// TIA Portal V20 export
FUNCTION_BLOCK "Sequence_3_NgPnP"   // FB245, LAD
AUTHOR : ERsystem_FA2_DH. Kim
// stored: IsIECCheckEnabled true, MemoryReserve 100, Namespace Unit1.Em4, SetENOAutomatically false
   VAR
      instSequenceLADStatus { ExternalWritable := 'False'} : "LAF_StatusLadSequence";
      instSequenceLADControl { ExternalWritable := 'False'} : "LAF_ControlLadSequence";
      statTonTime { ExternalWritable := 'False'} : Array[0..9999] of TON_TIME;
   END_VAR
   VAR_TEMP
      tempCustomerAction : Bool;   // Placeholder for possible actions
      tempDo_nothing_and_wait_for_init : Bool;   // Placeholder for doing nothing
      tempSafeStateCondition : Bool;   // Temp Condition for the equipment module to be in a safe state
   END_VAR
   VAR CONSTANT
      delayTime : Time := T#300ms;
      STEP_IDLE : DInt := 1;
      STEP_IMMEDIATE_STOP : DInt := 9001;   // Step executed when an immediate stop command is triggered for the sequence (i.e. when unit is in state aborting)
      JOB_1_STEP_01 : DInt := 101;
      JOB_1_STEP_10 : DInt := 110;
      JOB_1_STEP_20 : DInt := 120;
      JOB_1_STEP_30 : DInt := 130;
      JOB_1_STEP_80 : DInt := 180;
      JOB_1_STEP_81 : DInt := 181;
      JOB_1_STEP_90 : DInt := 190;
      JOB_2_STEP_01 : DInt := 201;
      JOB_2_STEP_10 : DInt := 210;
      JOB_2_STEP_20 : DInt := 220;
      JOB_2_STEP_30 : DInt := 230;
      JOB_2_STEP_31 : DInt := 231;
      JOB_2_STEP_40 : DInt := 240;
      JOB_2_STEP_80 : DInt := 280;
      JOB_2_STEP_90 : DInt := 290;
      JOB_3_STEP_01 : DInt := 301;
      JOB_3_STEP_20 : DInt := 320;
      JOB_3_STEP_30 : DInt := 330;
      JOB_3_STEP_40 : DInt := 340;
      JOB_3_STEP_90 : DInt := 390;
      FALSE : Bool := FALSE;
      TRUE : Bool := TRUE;
   END_VAR
   VAR_TEMP   // added for the SCL form of the ladder/FBD networks
      _w1 : Bool;
   END_VAR
BEGIN

REGION Network 1: BLOCK INFO HEADER
   // (company) / (C) Copyright (year)
   // ---------------------------------------------------------------------------------
   // Title:                             (Title of this block)
   // Comment/Function: (that is implemented in the block)
   // Library/Family:           (that the source is dedicated to)
   // Author:                        (department / person in charge / contact)
   // Target System:          (test system with FW version)
   // Engineering:              TIA Portal (SW version)
   // Restrictions:               (OB types, etc.)
   // Requirements:           (hardware, technological package, etc.)
   // ---------------------------------------------------------------------------------
   // Change log table:
   // Version          | Date             | Signature      | Expert in charge  | Changes applied ------------------------|----------------------|-------------------------|--------------------------------|-----------------------
   // 001.000.000 | yyyy-mm-dd | 0x00000000 | (name of expert) | First released version
END_REGION

REGION Network 2: DESCRIPTION
   // This is a template block provided by the Automation Framework. It can be used to create an own project.
   // The Block Info Header is prepared to put in your own data.
   // Description of the block could be added here and the docu created by Code2Docu.
END_REGION

REGION Network 3: ********************* CONTROL *************************
END_REGION

REGION Network 4: Sequence Control
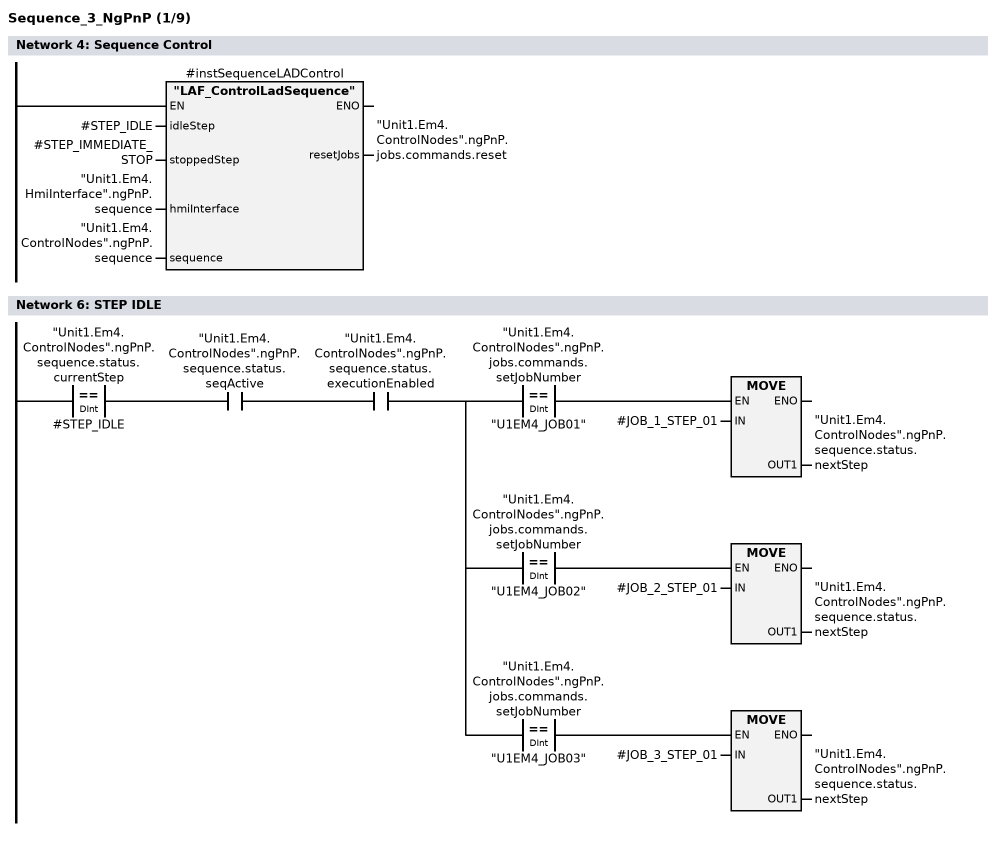
   RUNG wire#powerrail
      #instSequenceLADControl(idleStep := #STEP_IDLE, stoppedStep := #STEP_IMMEDIATE_STOP, hmiInterface := "Unit1.Em4.HmiInterface".ngPnP.sequence, sequence := "Unit1.Em4.ControlNodes".ngPnP.sequence, resetJobs => "Unit1.Em4.ControlNodes".ngPnP.jobs.commands.reset)
   END_RUNG
   // the same network as SCL:
   #instSequenceLADControl(idleStep := #STEP_IDLE,   // "LAF_ControlLadSequence"
                           stoppedStep := #STEP_IMMEDIATE_STOP,
                           hmiInterface := "Unit1.Em4.HmiInterface".ngPnP.sequence,
                           sequence := "Unit1.Em4.ControlNodes".ngPnP.sequence,
                           resetJobs => "Unit1.Em4.ControlNodes".ngPnP.jobs.commands.reset);
END_REGION

REGION Network 5: *************** JOB SELECT **************************
END_REGION

REGION Network 6: STEP IDLE
   RUNG wire#powerrail
      { S7_Templates := "SrcType := DInt" } EQ_Contact(in1 := "Unit1.Em4.ControlNodes".ngPnP.sequence.status.currentStep, in2 := #STEP_IDLE)
      Contact( "Unit1.Em4.ControlNodes".ngPnP.sequence.status.seqActive )
      Contact( "Unit1.Em4.ControlNodes".ngPnP.sequence.status.executionEnabled )
      wire#w1
      { S7_Templates := "SrcType := DInt" } EQ_Contact(in1 := "Unit1.Em4.ControlNodes".ngPnP.jobs.commands.setJobNumber, in2 := "U1EM4_JOB01")
      Move(in := #JOB_1_STEP_01, out1 => "Unit1.Em4.ControlNodes".ngPnP.sequence.status.nextStep)
   END_RUNG
   RUNG wire#w1
      { S7_Templates := "SrcType := DInt" } EQ_Contact(in1 := "Unit1.Em4.ControlNodes".ngPnP.jobs.commands.setJobNumber, in2 := "U1EM4_JOB02")
      Move(in := #JOB_2_STEP_01, out1 => "Unit1.Em4.ControlNodes".ngPnP.sequence.status.nextStep)
   END_RUNG
   RUNG wire#w1
      { S7_Templates := "SrcType := DInt" } EQ_Contact(in1 := "Unit1.Em4.ControlNodes".ngPnP.jobs.commands.setJobNumber, in2 := "U1EM4_JOB03")
      Move(in := #JOB_3_STEP_01, out1 => "Unit1.Em4.ControlNodes".ngPnP.sequence.status.nextStep)
   END_RUNG
   // the same network as SCL:
   #_w1 := ("Unit1.Em4.ControlNodes".ngPnP.sequence.status.currentStep = #STEP_IDLE) AND "Unit1.Em4.ControlNodes".ngPnP.sequence.status.seqActive AND "Unit1.Em4.ControlNodes".ngPnP.sequence.status.executionEnabled;
   IF #_w1 AND ("Unit1.Em4.ControlNodes".ngPnP.jobs.commands.setJobNumber = "U1EM4_JOB01") THEN
       "Unit1.Em4.ControlNodes".ngPnP.sequence.status.nextStep := #JOB_1_STEP_01;
   END_IF;
   IF #_w1 AND ("Unit1.Em4.ControlNodes".ngPnP.jobs.commands.setJobNumber = "U1EM4_JOB02") THEN
       "Unit1.Em4.ControlNodes".ngPnP.sequence.status.nextStep := #JOB_2_STEP_01;
   END_IF;
   IF #_w1 AND ("Unit1.Em4.ControlNodes".ngPnP.jobs.commands.setJobNumber = "U1EM4_JOB03") THEN
       "Unit1.Em4.ControlNodes".ngPnP.sequence.status.nextStep := #JOB_3_STEP_01;
   END_IF;
END_REGION

REGION Network 7: *************** JOB[1] EM HOMING ************************
END_REGION

REGION Network 8: Step[101] : JOB[1] Condition
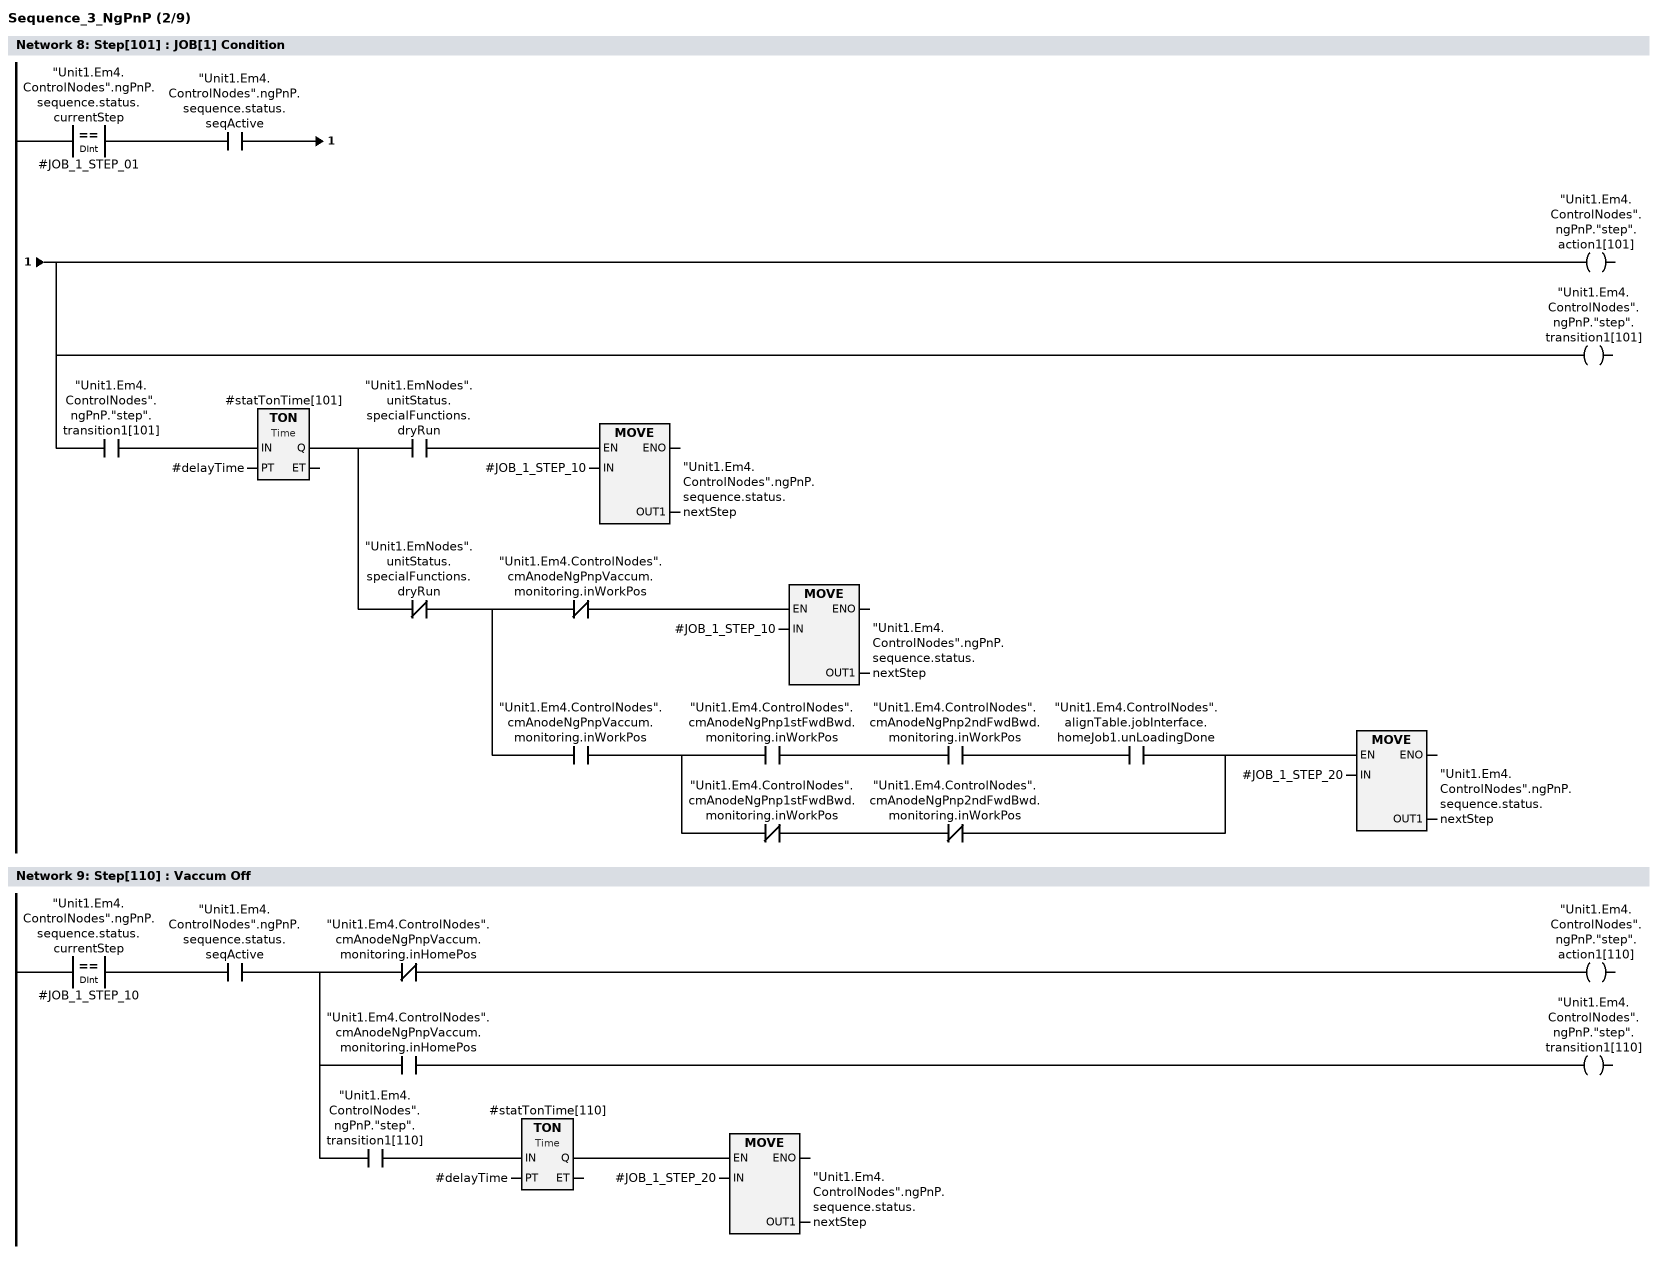
   RUNG wire#powerrail
      { S7_Templates := "SrcType := DInt" } EQ_Contact(in1 := "Unit1.Em4.ControlNodes".ngPnP.sequence.status.currentStep, in2 := #JOB_1_STEP_01)
      Contact( "Unit1.Em4.ControlNodes".ngPnP.sequence.status.seqActive )
      wire#w1
      Coil( "Unit1.Em4.ControlNodes".ngPnP."step".action1[101] )
   END_RUNG
   RUNG wire#w1
      Coil( "Unit1.Em4.ControlNodes".ngPnP."step".transition1[101] )
   END_RUNG
   RUNG wire#w1
      Contact( "Unit1.Em4.ControlNodes".ngPnP."step".transition1[101] )
      { S7_Templates := "time_type := Time" } #statTonTime[101].TON(pt := #delayTime, et =>)
      wire#w2
      Contact( "Unit1.EmNodes".unitStatus.specialFunctions.dryRun )
      Move(in := #JOB_1_STEP_10, out1 => "Unit1.Em4.ControlNodes".ngPnP.sequence.status.nextStep)
   END_RUNG
   RUNG wire#w2
      I_Contact( "Unit1.EmNodes".unitStatus.specialFunctions.dryRun )
      wire#w3
      I_Contact( "Unit1.Em4.ControlNodes".cmAnodeNgPnpVaccum.monitoring.inWorkPos )
      Move(in := #JOB_1_STEP_10, out1 => "Unit1.Em4.ControlNodes".ngPnP.sequence.status.nextStep)
   END_RUNG
   RUNG wire#w3
      Contact( "Unit1.Em4.ControlNodes".cmAnodeNgPnpVaccum.monitoring.inWorkPos )
      wire#w4
      Contact( "Unit1.Em4.ControlNodes".cmAnodeNgPnp1stFwdBwd.monitoring.inWorkPos )
      Contact( "Unit1.Em4.ControlNodes".cmAnodeNgPnp2ndFwdBwd.monitoring.inWorkPos )
      Contact( "Unit1.Em4.ControlNodes".alignTable.jobInterface.homeJob1.unLoadingDone )
      wire#w5
      Move(in := #JOB_1_STEP_20, out1 => "Unit1.Em4.ControlNodes".ngPnP.sequence.status.nextStep)
   END_RUNG
   RUNG wire#w4
      I_Contact( "Unit1.Em4.ControlNodes".cmAnodeNgPnp1stFwdBwd.monitoring.inWorkPos )
      I_Contact( "Unit1.Em4.ControlNodes".cmAnodeNgPnp2ndFwdBwd.monitoring.inWorkPos )
   END_RUNG wire#w5
   // the same network as SCL:
   "Unit1.Em4.ControlNodes".ngPnP."step".action1[101] := ("Unit1.Em4.ControlNodes".ngPnP.sequence.status.currentStep = #JOB_1_STEP_01) AND "Unit1.Em4.ControlNodes".ngPnP.sequence.status.seqActive;
   "Unit1.Em4.ControlNodes".ngPnP."step".transition1[101] := ("Unit1.Em4.ControlNodes".ngPnP.sequence.status.currentStep = #JOB_1_STEP_01) AND "Unit1.Em4.ControlNodes".ngPnP.sequence.status.seqActive;
   #statTonTime[101].TON(IN := ("Unit1.Em4.ControlNodes".ngPnP.sequence.status.currentStep = #JOB_1_STEP_01) AND "Unit1.Em4.ControlNodes".ngPnP.sequence.status.seqActive AND "Unit1.Em4.ControlNodes".ngPnP."step".transition1[101],
                         PT := #delayTime);
   IF #statTonTime[101].Q AND "Unit1.EmNodes".unitStatus.specialFunctions.dryRun THEN
       "Unit1.Em4.ControlNodes".ngPnP.sequence.status.nextStep := #JOB_1_STEP_10;
   END_IF;
   #_w1 := #statTonTime[101].Q AND NOT "Unit1.EmNodes".unitStatus.specialFunctions.dryRun;
   IF #_w1 AND NOT "Unit1.Em4.ControlNodes".cmAnodeNgPnpVaccum.monitoring.inWorkPos THEN
       "Unit1.Em4.ControlNodes".ngPnP.sequence.status.nextStep := #JOB_1_STEP_10;
   END_IF;
   IF #_w1 AND "Unit1.Em4.ControlNodes".cmAnodeNgPnpVaccum.monitoring.inWorkPos AND (("Unit1.Em4.ControlNodes".cmAnodeNgPnp1stFwdBwd.monitoring.inWorkPos AND "Unit1.Em4.ControlNodes".cmAnodeNgPnp2ndFwdBwd.monitoring.inWorkPos AND "Unit1.Em4.ControlNodes".alignTable.jobInterface.homeJob1.unLoadingDone) OR (NOT "Unit1.Em4.ControlNodes".cmAnodeNgPnp1stFwdBwd.monitoring.inWorkPos AND NOT "Unit1.Em4.ControlNodes".cmAnodeNgPnp2ndFwdBwd.monitoring.inWorkPos)) THEN
       "Unit1.Em4.ControlNodes".ngPnP.sequence.status.nextStep := #JOB_1_STEP_20;
   END_IF;
END_REGION

REGION Network 9: Step[110] : Vaccum Off
   RUNG wire#powerrail
      { S7_Templates := "SrcType := DInt" } EQ_Contact(in1 := "Unit1.Em4.ControlNodes".ngPnP.sequence.status.currentStep, in2 := #JOB_1_STEP_10)
      Contact( "Unit1.Em4.ControlNodes".ngPnP.sequence.status.seqActive )
      wire#w1
      I_Contact( "Unit1.Em4.ControlNodes".cmAnodeNgPnpVaccum.monitoring.inHomePos )
      Coil( "Unit1.Em4.ControlNodes".ngPnP."step".action1[110] )
   END_RUNG
   RUNG wire#w1
      Contact( "Unit1.Em4.ControlNodes".cmAnodeNgPnpVaccum.monitoring.inHomePos )
      Coil( "Unit1.Em4.ControlNodes".ngPnP."step".transition1[110] )
   END_RUNG
   RUNG wire#w1
      Contact( "Unit1.Em4.ControlNodes".ngPnP."step".transition1[110] )
      { S7_Templates := "time_type := Time" } #statTonTime[110].TON(pt := #delayTime, et =>)
      Move(in := #JOB_1_STEP_20, out1 => "Unit1.Em4.ControlNodes".ngPnP.sequence.status.nextStep)
   END_RUNG
   // the same network as SCL:
   #_w1 := ("Unit1.Em4.ControlNodes".ngPnP.sequence.status.currentStep = #JOB_1_STEP_10) AND "Unit1.Em4.ControlNodes".ngPnP.sequence.status.seqActive;
   "Unit1.Em4.ControlNodes".ngPnP."step".action1[110] := #_w1 AND NOT "Unit1.Em4.ControlNodes".cmAnodeNgPnpVaccum.monitoring.inHomePos;
   "Unit1.Em4.ControlNodes".ngPnP."step".transition1[110] := #_w1 AND "Unit1.Em4.ControlNodes".cmAnodeNgPnpVaccum.monitoring.inHomePos;
   #statTonTime[110].TON(IN := #_w1 AND "Unit1.Em4.ControlNodes".ngPnP."step".transition1[110],
                         PT := #delayTime);
   IF #statTonTime[110].Q THEN
       "Unit1.Em4.ControlNodes".ngPnP.sequence.status.nextStep := #JOB_1_STEP_20;
   END_IF;
END_REGION

REGION Network 10: Step[120] : NG P&P Up
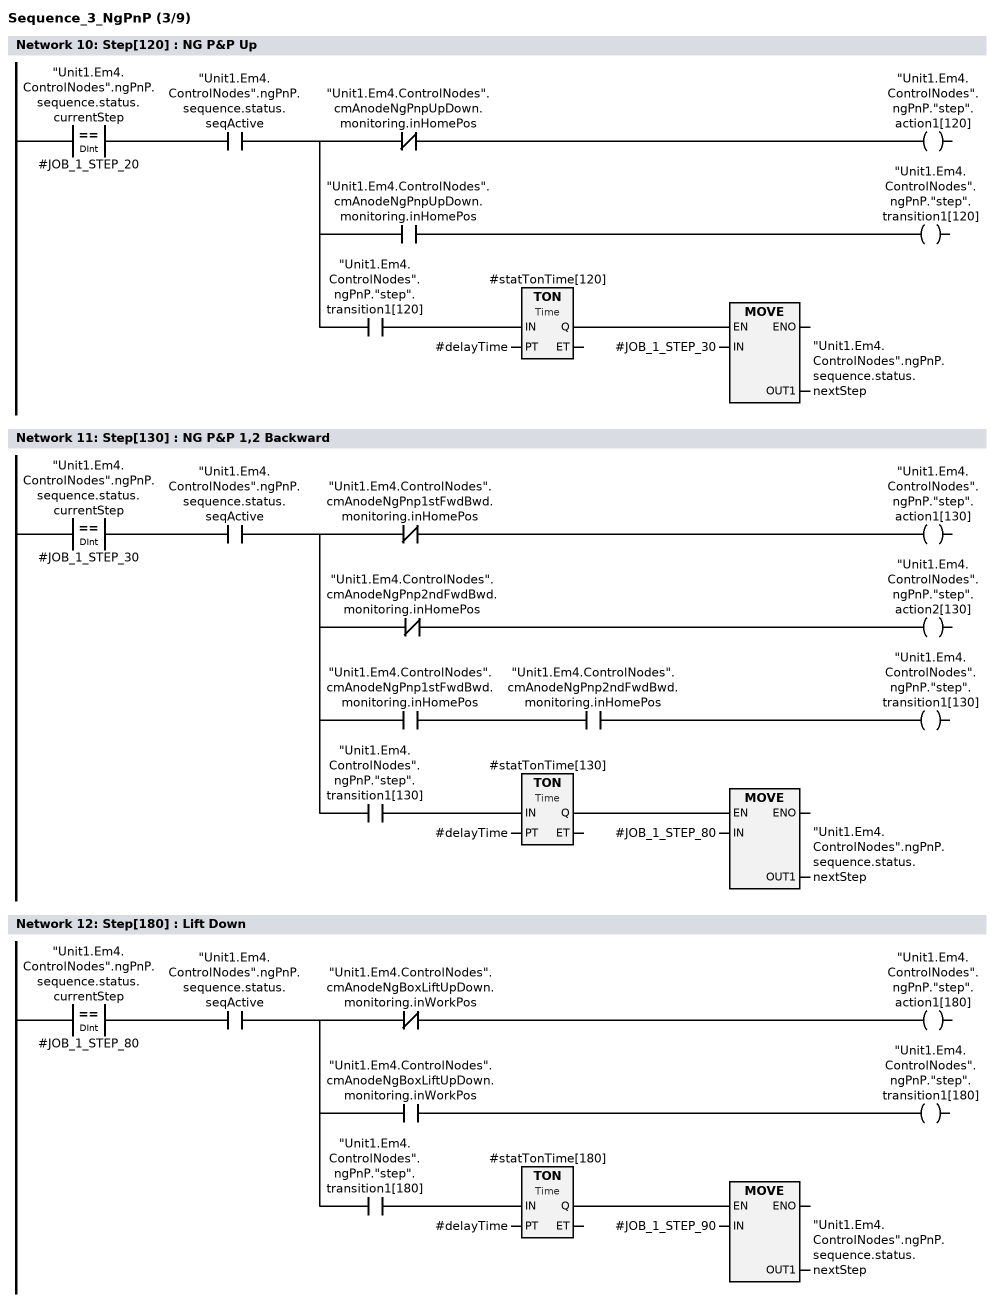
   RUNG wire#powerrail
      { S7_Templates := "SrcType := DInt" } EQ_Contact(in1 := "Unit1.Em4.ControlNodes".ngPnP.sequence.status.currentStep, in2 := #JOB_1_STEP_20)
      Contact( "Unit1.Em4.ControlNodes".ngPnP.sequence.status.seqActive )
      wire#w1
      I_Contact( "Unit1.Em4.ControlNodes".cmAnodeNgPnpUpDown.monitoring.inHomePos )
      Coil( "Unit1.Em4.ControlNodes".ngPnP."step".action1[120] )
   END_RUNG
   RUNG wire#w1
      Contact( "Unit1.Em4.ControlNodes".cmAnodeNgPnpUpDown.monitoring.inHomePos )
      Coil( "Unit1.Em4.ControlNodes".ngPnP."step".transition1[120] )
   END_RUNG
   RUNG wire#w1
      Contact( "Unit1.Em4.ControlNodes".ngPnP."step".transition1[120] )
      { S7_Templates := "time_type := Time" } #statTonTime[120].TON(pt := #delayTime, et =>)
      Move(in := #JOB_1_STEP_30, out1 => "Unit1.Em4.ControlNodes".ngPnP.sequence.status.nextStep)
   END_RUNG
   // the same network as SCL:
   #_w1 := ("Unit1.Em4.ControlNodes".ngPnP.sequence.status.currentStep = #JOB_1_STEP_20) AND "Unit1.Em4.ControlNodes".ngPnP.sequence.status.seqActive;
   "Unit1.Em4.ControlNodes".ngPnP."step".action1[120] := #_w1 AND NOT "Unit1.Em4.ControlNodes".cmAnodeNgPnpUpDown.monitoring.inHomePos;
   "Unit1.Em4.ControlNodes".ngPnP."step".transition1[120] := #_w1 AND "Unit1.Em4.ControlNodes".cmAnodeNgPnpUpDown.monitoring.inHomePos;
   #statTonTime[120].TON(IN := #_w1 AND "Unit1.Em4.ControlNodes".ngPnP."step".transition1[120],
                         PT := #delayTime);
   IF #statTonTime[120].Q THEN
       "Unit1.Em4.ControlNodes".ngPnP.sequence.status.nextStep := #JOB_1_STEP_30;
   END_IF;
END_REGION

REGION Network 11: Step[130] : NG P&P 1,2 Backward
   RUNG wire#powerrail
      { S7_Templates := "SrcType := DInt" } EQ_Contact(in1 := "Unit1.Em4.ControlNodes".ngPnP.sequence.status.currentStep, in2 := #JOB_1_STEP_30)
      Contact( "Unit1.Em4.ControlNodes".ngPnP.sequence.status.seqActive )
      wire#w1
      I_Contact( "Unit1.Em4.ControlNodes".cmAnodeNgPnp1stFwdBwd.monitoring.inHomePos )
      Coil( "Unit1.Em4.ControlNodes".ngPnP."step".action1[130] )
   END_RUNG
   RUNG wire#w1
      I_Contact( "Unit1.Em4.ControlNodes".cmAnodeNgPnp2ndFwdBwd.monitoring.inHomePos )
      Coil( "Unit1.Em4.ControlNodes".ngPnP."step".action2[130] )
   END_RUNG
   RUNG wire#w1
      Contact( "Unit1.Em4.ControlNodes".cmAnodeNgPnp1stFwdBwd.monitoring.inHomePos )
      Contact( "Unit1.Em4.ControlNodes".cmAnodeNgPnp2ndFwdBwd.monitoring.inHomePos )
      Coil( "Unit1.Em4.ControlNodes".ngPnP."step".transition1[130] )
   END_RUNG
   RUNG wire#w1
      Contact( "Unit1.Em4.ControlNodes".ngPnP."step".transition1[130] )
      { S7_Templates := "time_type := Time" } #statTonTime[130].TON(pt := #delayTime, et =>)
      Move(in := #JOB_1_STEP_80, out1 => "Unit1.Em4.ControlNodes".ngPnP.sequence.status.nextStep)
   END_RUNG
   // the same network as SCL:
   #_w1 := ("Unit1.Em4.ControlNodes".ngPnP.sequence.status.currentStep = #JOB_1_STEP_30) AND "Unit1.Em4.ControlNodes".ngPnP.sequence.status.seqActive;
   "Unit1.Em4.ControlNodes".ngPnP."step".action1[130] := #_w1 AND NOT "Unit1.Em4.ControlNodes".cmAnodeNgPnp1stFwdBwd.monitoring.inHomePos;
   "Unit1.Em4.ControlNodes".ngPnP."step".action2[130] := #_w1 AND NOT "Unit1.Em4.ControlNodes".cmAnodeNgPnp2ndFwdBwd.monitoring.inHomePos;
   "Unit1.Em4.ControlNodes".ngPnP."step".transition1[130] := #_w1 AND "Unit1.Em4.ControlNodes".cmAnodeNgPnp1stFwdBwd.monitoring.inHomePos AND "Unit1.Em4.ControlNodes".cmAnodeNgPnp2ndFwdBwd.monitoring.inHomePos;
   #statTonTime[130].TON(IN := #_w1 AND "Unit1.Em4.ControlNodes".ngPnP."step".transition1[130],
                         PT := #delayTime);
   IF #statTonTime[130].Q THEN
       "Unit1.Em4.ControlNodes".ngPnP.sequence.status.nextStep := #JOB_1_STEP_80;
   END_IF;
END_REGION

REGION Network 12: Step[180] : Lift Down
   RUNG wire#powerrail
      { S7_Templates := "SrcType := DInt" } EQ_Contact(in1 := "Unit1.Em4.ControlNodes".ngPnP.sequence.status.currentStep, in2 := #JOB_1_STEP_80)
      Contact( "Unit1.Em4.ControlNodes".ngPnP.sequence.status.seqActive )
      wire#w1
      I_Contact( "Unit1.Em4.ControlNodes".cmAnodeNgBoxLiftUpDown.monitoring.inWorkPos )
      Coil( "Unit1.Em4.ControlNodes".ngPnP."step".action1[180] )
   END_RUNG
   RUNG wire#w1
      Contact( "Unit1.Em4.ControlNodes".cmAnodeNgBoxLiftUpDown.monitoring.inWorkPos )
      Coil( "Unit1.Em4.ControlNodes".ngPnP."step".transition1[180] )
   END_RUNG
   RUNG wire#w1
      Contact( "Unit1.Em4.ControlNodes".ngPnP."step".transition1[180] )
      { S7_Templates := "time_type := Time" } #statTonTime[180].TON(pt := #delayTime, et =>)
      Move(in := #JOB_1_STEP_90, out1 => "Unit1.Em4.ControlNodes".ngPnP.sequence.status.nextStep)
   END_RUNG
   // the same network as SCL:
   #_w1 := ("Unit1.Em4.ControlNodes".ngPnP.sequence.status.currentStep = #JOB_1_STEP_80) AND "Unit1.Em4.ControlNodes".ngPnP.sequence.status.seqActive;
   "Unit1.Em4.ControlNodes".ngPnP."step".action1[180] := #_w1 AND NOT "Unit1.Em4.ControlNodes".cmAnodeNgBoxLiftUpDown.monitoring.inWorkPos;
   "Unit1.Em4.ControlNodes".ngPnP."step".transition1[180] := #_w1 AND "Unit1.Em4.ControlNodes".cmAnodeNgBoxLiftUpDown.monitoring.inWorkPos;
   #statTonTime[180].TON(IN := #_w1 AND "Unit1.Em4.ControlNodes".ngPnP."step".transition1[180],
                         PT := #delayTime);
   IF #statTonTime[180].Q THEN
       "Unit1.Em4.ControlNodes".ngPnP.sequence.status.nextStep := #JOB_1_STEP_90;
   END_IF;
END_REGION

REGION Network 13: Step[190] : JOB[1] Step End
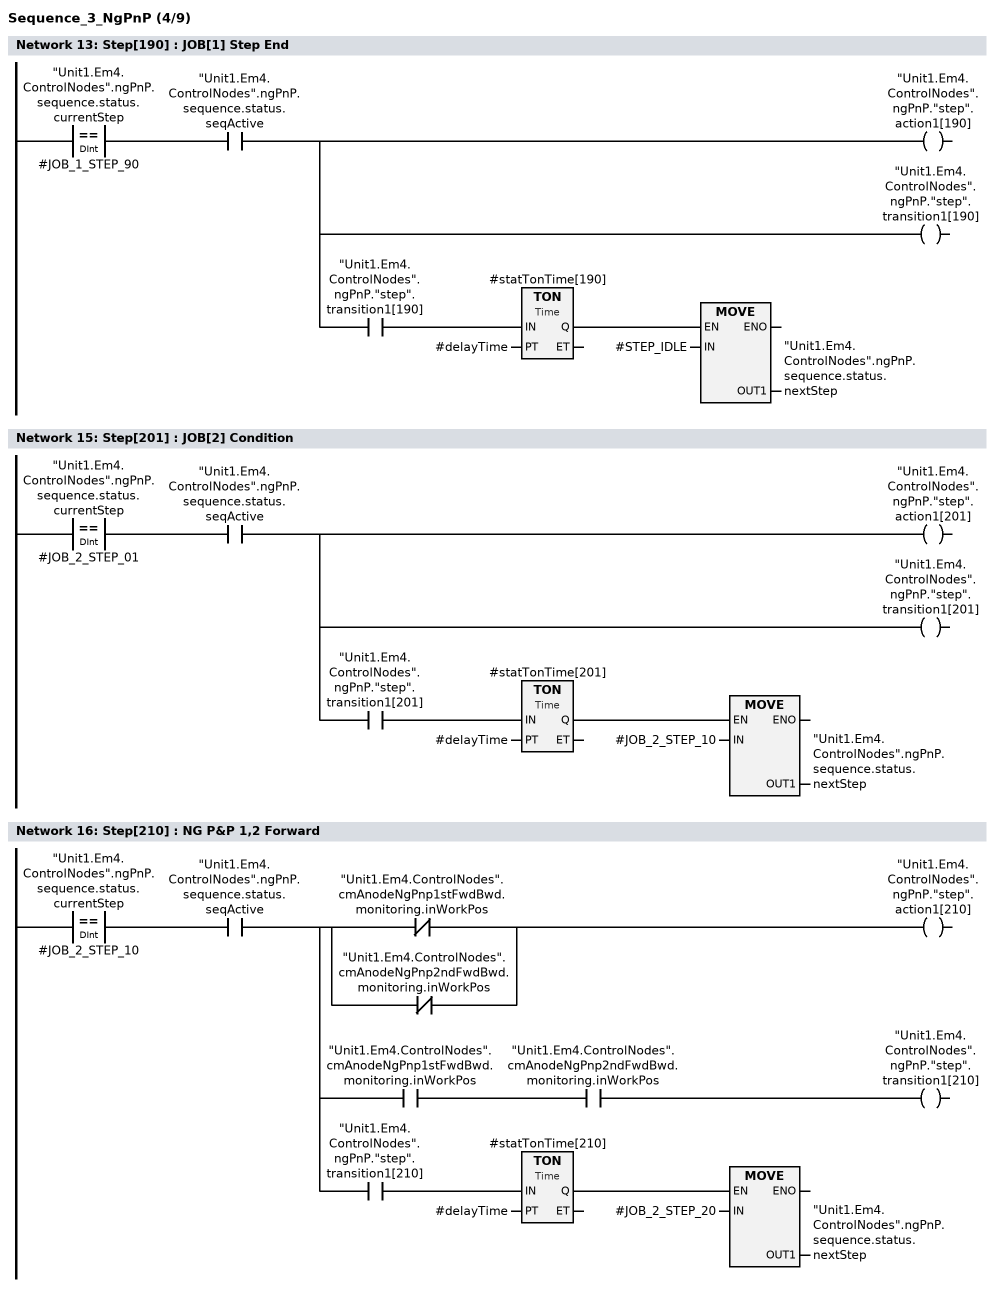
   RUNG wire#powerrail
      { S7_Templates := "SrcType := DInt" } EQ_Contact(in1 := "Unit1.Em4.ControlNodes".ngPnP.sequence.status.currentStep, in2 := #JOB_1_STEP_90)
      Contact( "Unit1.Em4.ControlNodes".ngPnP.sequence.status.seqActive )
      wire#w1
      Coil( "Unit1.Em4.ControlNodes".ngPnP."step".action1[190] )
   END_RUNG
   RUNG wire#w1
      Coil( "Unit1.Em4.ControlNodes".ngPnP."step".transition1[190] )
   END_RUNG
   RUNG wire#w1
      Contact( "Unit1.Em4.ControlNodes".ngPnP."step".transition1[190] )
      { S7_Templates := "time_type := Time" } #statTonTime[190].TON(pt := #delayTime, et =>)
      Move(in := #STEP_IDLE, out1 => "Unit1.Em4.ControlNodes".ngPnP.sequence.status.nextStep)
   END_RUNG
   // the same network as SCL:
   "Unit1.Em4.ControlNodes".ngPnP."step".action1[190] := ("Unit1.Em4.ControlNodes".ngPnP.sequence.status.currentStep = #JOB_1_STEP_90) AND "Unit1.Em4.ControlNodes".ngPnP.sequence.status.seqActive;
   "Unit1.Em4.ControlNodes".ngPnP."step".transition1[190] := ("Unit1.Em4.ControlNodes".ngPnP.sequence.status.currentStep = #JOB_1_STEP_90) AND "Unit1.Em4.ControlNodes".ngPnP.sequence.status.seqActive;
   #statTonTime[190].TON(IN := ("Unit1.Em4.ControlNodes".ngPnP.sequence.status.currentStep = #JOB_1_STEP_90) AND "Unit1.Em4.ControlNodes".ngPnP.sequence.status.seqActive AND "Unit1.Em4.ControlNodes".ngPnP."step".transition1[190],
                         PT := #delayTime);
   IF #statTonTime[190].Q THEN "Unit1.Em4.ControlNodes".ngPnP.sequence.status.nextStep := #STEP_IDLE; END_IF;
END_REGION

REGION Network 14: *************** JOB[2] Loading ************************
END_REGION

REGION Network 15: Step[201] : JOB[2] Condition
   RUNG wire#powerrail
      { S7_Templates := "SrcType := DInt" } EQ_Contact(in1 := "Unit1.Em4.ControlNodes".ngPnP.sequence.status.currentStep, in2 := #JOB_2_STEP_01)
      Contact( "Unit1.Em4.ControlNodes".ngPnP.sequence.status.seqActive )
      wire#w1
      Coil( "Unit1.Em4.ControlNodes".ngPnP."step".action1[201] )
   END_RUNG
   RUNG wire#w1
      Coil( "Unit1.Em4.ControlNodes".ngPnP."step".transition1[201] )
   END_RUNG
   RUNG wire#w1
      Contact( "Unit1.Em4.ControlNodes".ngPnP."step".transition1[201] )
      { S7_Templates := "time_type := Time" } #statTonTime[201].TON(pt := #delayTime, et =>)
      Move(in := #JOB_2_STEP_10, out1 => "Unit1.Em4.ControlNodes".ngPnP.sequence.status.nextStep)
   END_RUNG
   // the same network as SCL:
   "Unit1.Em4.ControlNodes".ngPnP."step".action1[201] := ("Unit1.Em4.ControlNodes".ngPnP.sequence.status.currentStep = #JOB_2_STEP_01) AND "Unit1.Em4.ControlNodes".ngPnP.sequence.status.seqActive;
   "Unit1.Em4.ControlNodes".ngPnP."step".transition1[201] := ("Unit1.Em4.ControlNodes".ngPnP.sequence.status.currentStep = #JOB_2_STEP_01) AND "Unit1.Em4.ControlNodes".ngPnP.sequence.status.seqActive;
   #statTonTime[201].TON(IN := ("Unit1.Em4.ControlNodes".ngPnP.sequence.status.currentStep = #JOB_2_STEP_01) AND "Unit1.Em4.ControlNodes".ngPnP.sequence.status.seqActive AND "Unit1.Em4.ControlNodes".ngPnP."step".transition1[201],
                         PT := #delayTime);
   IF #statTonTime[201].Q THEN
       "Unit1.Em4.ControlNodes".ngPnP.sequence.status.nextStep := #JOB_2_STEP_10;
   END_IF;
END_REGION

REGION Network 16: Step[210] : NG P&P 1,2 Forward
   RUNG wire#powerrail
      { S7_Templates := "SrcType := DInt" } EQ_Contact(in1 := "Unit1.Em4.ControlNodes".ngPnP.sequence.status.currentStep, in2 := #JOB_2_STEP_10)
      Contact( "Unit1.Em4.ControlNodes".ngPnP.sequence.status.seqActive )
      wire#w1
      I_Contact( "Unit1.Em4.ControlNodes".cmAnodeNgPnp1stFwdBwd.monitoring.inWorkPos )
      wire#w2
      Coil( "Unit1.Em4.ControlNodes".ngPnP."step".action1[210] )
   END_RUNG
   RUNG wire#w1
      I_Contact( "Unit1.Em4.ControlNodes".cmAnodeNgPnp2ndFwdBwd.monitoring.inWorkPos )
   END_RUNG wire#w2
   RUNG wire#w1
      Contact( "Unit1.Em4.ControlNodes".cmAnodeNgPnp1stFwdBwd.monitoring.inWorkPos )
      Contact( "Unit1.Em4.ControlNodes".cmAnodeNgPnp2ndFwdBwd.monitoring.inWorkPos )
      Coil( "Unit1.Em4.ControlNodes".ngPnP."step".transition1[210] )
   END_RUNG
   RUNG wire#w1
      Contact( "Unit1.Em4.ControlNodes".ngPnP."step".transition1[210] )
      { S7_Templates := "time_type := Time" } #statTonTime[210].TON(pt := #delayTime, et =>)
      Move(in := #JOB_2_STEP_20, out1 => "Unit1.Em4.ControlNodes".ngPnP.sequence.status.nextStep)
   END_RUNG
   // the same network as SCL:
   #_w1 := ("Unit1.Em4.ControlNodes".ngPnP.sequence.status.currentStep = #JOB_2_STEP_10) AND "Unit1.Em4.ControlNodes".ngPnP.sequence.status.seqActive;
   "Unit1.Em4.ControlNodes".ngPnP."step".action1[210] := #_w1 AND (NOT "Unit1.Em4.ControlNodes".cmAnodeNgPnp1stFwdBwd.monitoring.inWorkPos OR NOT "Unit1.Em4.ControlNodes".cmAnodeNgPnp2ndFwdBwd.monitoring.inWorkPos);
   "Unit1.Em4.ControlNodes".ngPnP."step".transition1[210] := #_w1 AND "Unit1.Em4.ControlNodes".cmAnodeNgPnp1stFwdBwd.monitoring.inWorkPos AND "Unit1.Em4.ControlNodes".cmAnodeNgPnp2ndFwdBwd.monitoring.inWorkPos;
   #statTonTime[210].TON(IN := #_w1 AND "Unit1.Em4.ControlNodes".ngPnP."step".transition1[210],
                         PT := #delayTime);
   IF #statTonTime[210].Q THEN
       "Unit1.Em4.ControlNodes".ngPnP.sequence.status.nextStep := #JOB_2_STEP_20;
   END_IF;
END_REGION

REGION Network 17: Step[220] : NG P&P Down
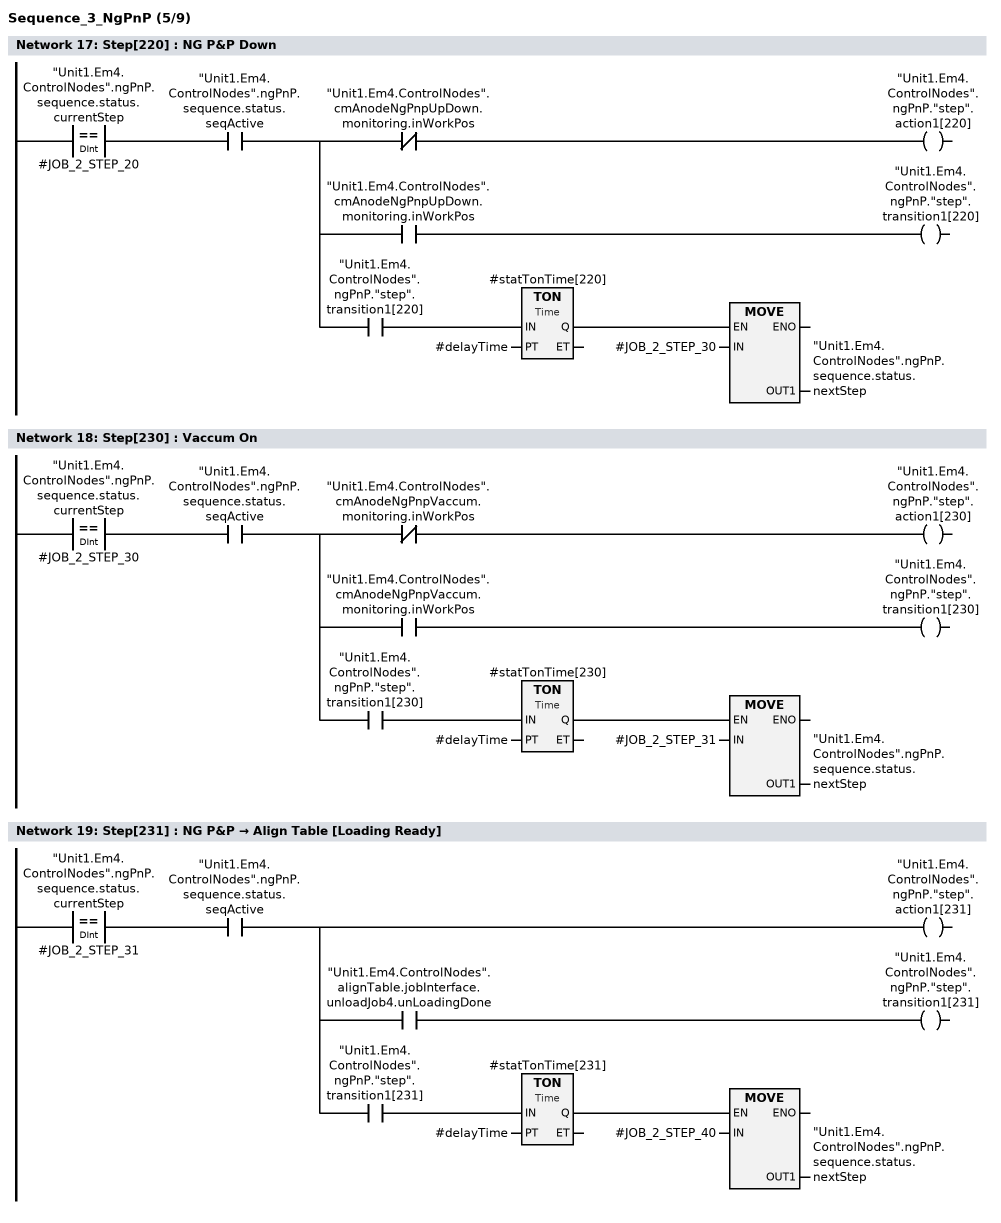
   RUNG wire#powerrail
      { S7_Templates := "SrcType := DInt" } EQ_Contact(in1 := "Unit1.Em4.ControlNodes".ngPnP.sequence.status.currentStep, in2 := #JOB_2_STEP_20)
      Contact( "Unit1.Em4.ControlNodes".ngPnP.sequence.status.seqActive )
      wire#w1
      I_Contact( "Unit1.Em4.ControlNodes".cmAnodeNgPnpUpDown.monitoring.inWorkPos )
      Coil( "Unit1.Em4.ControlNodes".ngPnP."step".action1[220] )
   END_RUNG
   RUNG wire#w1
      Contact( "Unit1.Em4.ControlNodes".cmAnodeNgPnpUpDown.monitoring.inWorkPos )
      Coil( "Unit1.Em4.ControlNodes".ngPnP."step".transition1[220] )
   END_RUNG
   RUNG wire#w1
      Contact( "Unit1.Em4.ControlNodes".ngPnP."step".transition1[220] )
      { S7_Templates := "time_type := Time" } #statTonTime[220].TON(pt := #delayTime, et =>)
      Move(in := #JOB_2_STEP_30, out1 => "Unit1.Em4.ControlNodes".ngPnP.sequence.status.nextStep)
   END_RUNG
   // the same network as SCL:
   #_w1 := ("Unit1.Em4.ControlNodes".ngPnP.sequence.status.currentStep = #JOB_2_STEP_20) AND "Unit1.Em4.ControlNodes".ngPnP.sequence.status.seqActive;
   "Unit1.Em4.ControlNodes".ngPnP."step".action1[220] := #_w1 AND NOT "Unit1.Em4.ControlNodes".cmAnodeNgPnpUpDown.monitoring.inWorkPos;
   "Unit1.Em4.ControlNodes".ngPnP."step".transition1[220] := #_w1 AND "Unit1.Em4.ControlNodes".cmAnodeNgPnpUpDown.monitoring.inWorkPos;
   #statTonTime[220].TON(IN := #_w1 AND "Unit1.Em4.ControlNodes".ngPnP."step".transition1[220],
                         PT := #delayTime);
   IF #statTonTime[220].Q THEN
       "Unit1.Em4.ControlNodes".ngPnP.sequence.status.nextStep := #JOB_2_STEP_30;
   END_IF;
END_REGION

REGION Network 18: Step[230] : Vaccum On
   RUNG wire#powerrail
      { S7_Templates := "SrcType := DInt" } EQ_Contact(in1 := "Unit1.Em4.ControlNodes".ngPnP.sequence.status.currentStep, in2 := #JOB_2_STEP_30)
      Contact( "Unit1.Em4.ControlNodes".ngPnP.sequence.status.seqActive )
      wire#w1
      I_Contact( "Unit1.Em4.ControlNodes".cmAnodeNgPnpVaccum.monitoring.inWorkPos )
      Coil( "Unit1.Em4.ControlNodes".ngPnP."step".action1[230] )
   END_RUNG
   RUNG wire#w1
      Contact( "Unit1.Em4.ControlNodes".cmAnodeNgPnpVaccum.monitoring.inWorkPos )
      Coil( "Unit1.Em4.ControlNodes".ngPnP."step".transition1[230] )
   END_RUNG
   RUNG wire#w1
      Contact( "Unit1.Em4.ControlNodes".ngPnP."step".transition1[230] )
      { S7_Templates := "time_type := Time" } #statTonTime[230].TON(pt := #delayTime, et =>)
      Move(in := #JOB_2_STEP_31, out1 => "Unit1.Em4.ControlNodes".ngPnP.sequence.status.nextStep)
   END_RUNG
   // the same network as SCL:
   #_w1 := ("Unit1.Em4.ControlNodes".ngPnP.sequence.status.currentStep = #JOB_2_STEP_30) AND "Unit1.Em4.ControlNodes".ngPnP.sequence.status.seqActive;
   "Unit1.Em4.ControlNodes".ngPnP."step".action1[230] := #_w1 AND NOT "Unit1.Em4.ControlNodes".cmAnodeNgPnpVaccum.monitoring.inWorkPos;
   "Unit1.Em4.ControlNodes".ngPnP."step".transition1[230] := #_w1 AND "Unit1.Em4.ControlNodes".cmAnodeNgPnpVaccum.monitoring.inWorkPos;
   #statTonTime[230].TON(IN := #_w1 AND "Unit1.Em4.ControlNodes".ngPnP."step".transition1[230],
                         PT := #delayTime);
   IF #statTonTime[230].Q THEN
       "Unit1.Em4.ControlNodes".ngPnP.sequence.status.nextStep := #JOB_2_STEP_31;
   END_IF;
END_REGION

REGION Network 19: Step[231] : NG P&P → Align Table [Loading Ready]
   RUNG wire#powerrail
      { S7_Templates := "SrcType := DInt" } EQ_Contact(in1 := "Unit1.Em4.ControlNodes".ngPnP.sequence.status.currentStep, in2 := #JOB_2_STEP_31)
      Contact( "Unit1.Em4.ControlNodes".ngPnP.sequence.status.seqActive )
      wire#w1
      Coil( "Unit1.Em4.ControlNodes".ngPnP."step".action1[231] )
   END_RUNG
   RUNG wire#w1
      Contact( "Unit1.Em4.ControlNodes".alignTable.jobInterface.unloadJob4.unLoadingDone )
      Coil( "Unit1.Em4.ControlNodes".ngPnP."step".transition1[231] )
   END_RUNG
   RUNG wire#w1
      Contact( "Unit1.Em4.ControlNodes".ngPnP."step".transition1[231] )
      { S7_Templates := "time_type := Time" } #statTonTime[231].TON(pt := #delayTime, et =>)
      Move(in := #JOB_2_STEP_40, out1 => "Unit1.Em4.ControlNodes".ngPnP.sequence.status.nextStep)
   END_RUNG
   // the same network as SCL:
   "Unit1.Em4.ControlNodes".ngPnP."step".action1[231] := ("Unit1.Em4.ControlNodes".ngPnP.sequence.status.currentStep = #JOB_2_STEP_31) AND "Unit1.Em4.ControlNodes".ngPnP.sequence.status.seqActive;
   "Unit1.Em4.ControlNodes".ngPnP."step".transition1[231] := ("Unit1.Em4.ControlNodes".ngPnP.sequence.status.currentStep = #JOB_2_STEP_31) AND "Unit1.Em4.ControlNodes".ngPnP.sequence.status.seqActive AND "Unit1.Em4.ControlNodes".alignTable.jobInterface.unloadJob4.unLoadingDone;
   #statTonTime[231].TON(IN := ("Unit1.Em4.ControlNodes".ngPnP.sequence.status.currentStep = #JOB_2_STEP_31) AND "Unit1.Em4.ControlNodes".ngPnP.sequence.status.seqActive AND "Unit1.Em4.ControlNodes".ngPnP."step".transition1[231],
                         PT := #delayTime);
   IF #statTonTime[231].Q THEN
       "Unit1.Em4.ControlNodes".ngPnP.sequence.status.nextStep := #JOB_2_STEP_40;
   END_IF;
END_REGION

REGION Network 20: Step[240] : NG P&P Up
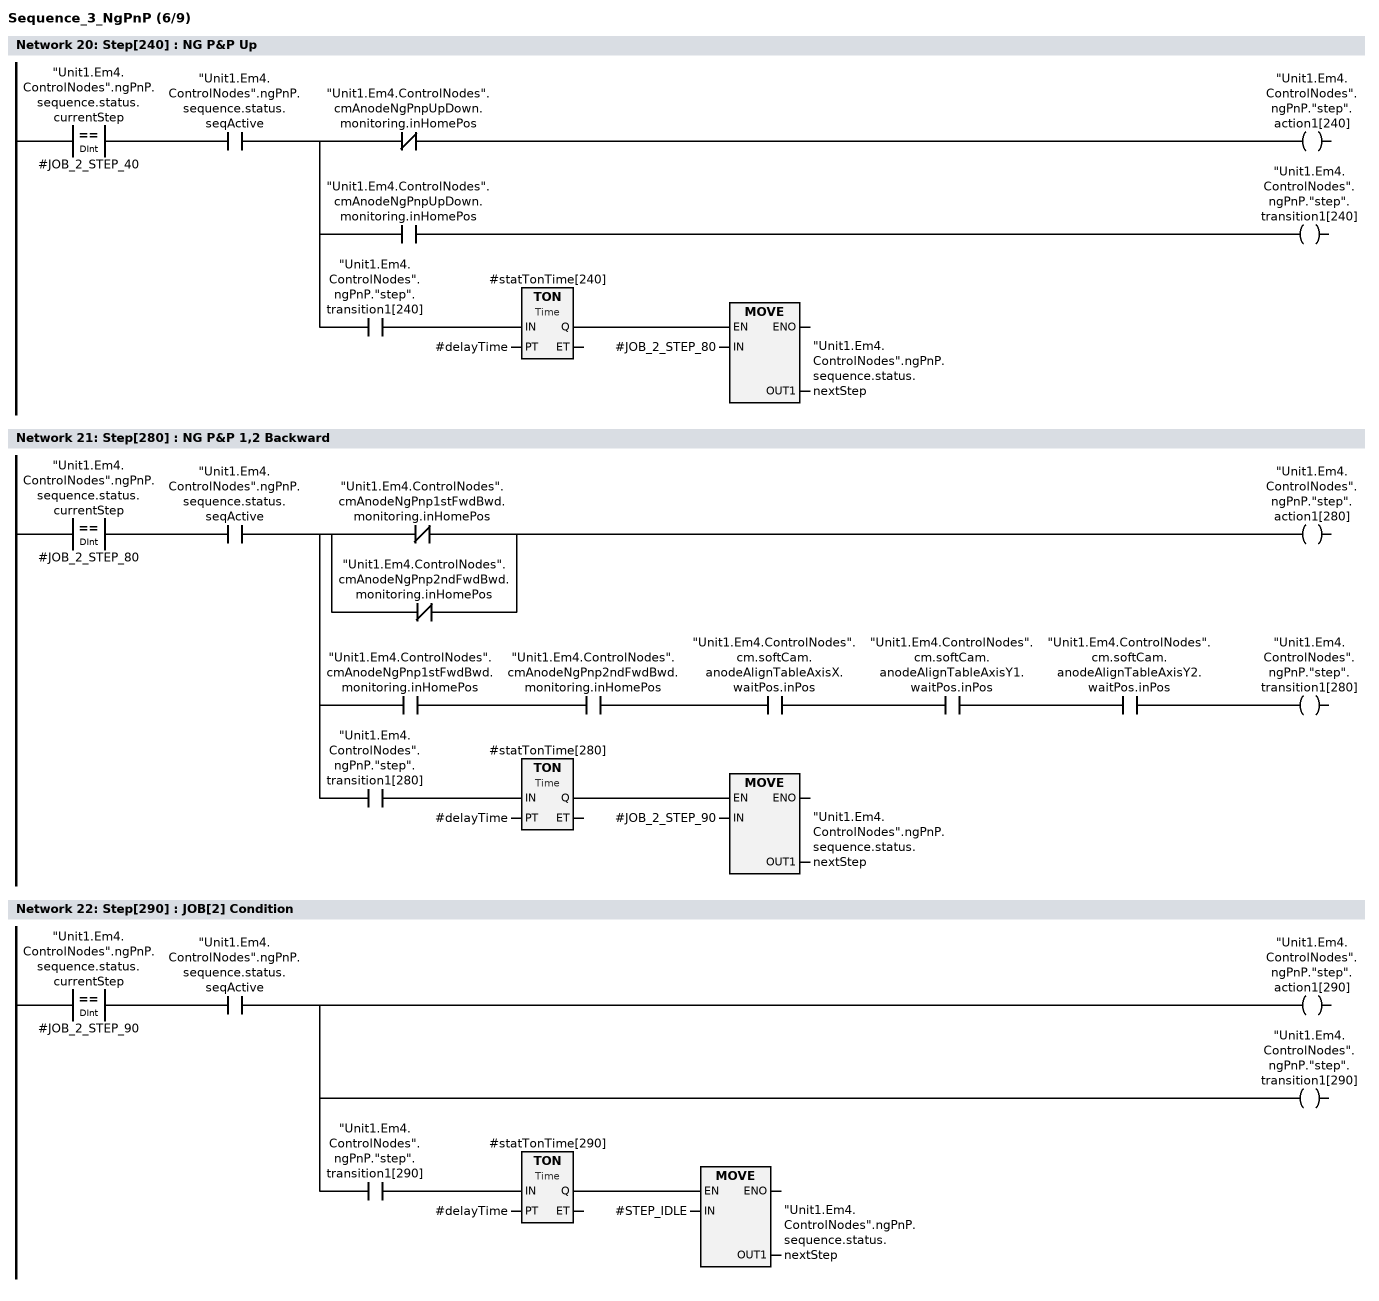
   RUNG wire#powerrail
      { S7_Templates := "SrcType := DInt" } EQ_Contact(in1 := "Unit1.Em4.ControlNodes".ngPnP.sequence.status.currentStep, in2 := #JOB_2_STEP_40)
      Contact( "Unit1.Em4.ControlNodes".ngPnP.sequence.status.seqActive )
      wire#w1
      I_Contact( "Unit1.Em4.ControlNodes".cmAnodeNgPnpUpDown.monitoring.inHomePos )
      Coil( "Unit1.Em4.ControlNodes".ngPnP."step".action1[240] )
   END_RUNG
   RUNG wire#w1
      Contact( "Unit1.Em4.ControlNodes".cmAnodeNgPnpUpDown.monitoring.inHomePos )
      Coil( "Unit1.Em4.ControlNodes".ngPnP."step".transition1[240] )
   END_RUNG
   RUNG wire#w1
      Contact( "Unit1.Em4.ControlNodes".ngPnP."step".transition1[240] )
      { S7_Templates := "time_type := Time" } #statTonTime[240].TON(pt := #delayTime, et =>)
      Move(in := #JOB_2_STEP_80, out1 => "Unit1.Em4.ControlNodes".ngPnP.sequence.status.nextStep)
   END_RUNG
   // the same network as SCL:
   #_w1 := ("Unit1.Em4.ControlNodes".ngPnP.sequence.status.currentStep = #JOB_2_STEP_40) AND "Unit1.Em4.ControlNodes".ngPnP.sequence.status.seqActive;
   "Unit1.Em4.ControlNodes".ngPnP."step".action1[240] := #_w1 AND NOT "Unit1.Em4.ControlNodes".cmAnodeNgPnpUpDown.monitoring.inHomePos;
   "Unit1.Em4.ControlNodes".ngPnP."step".transition1[240] := #_w1 AND "Unit1.Em4.ControlNodes".cmAnodeNgPnpUpDown.monitoring.inHomePos;
   #statTonTime[240].TON(IN := #_w1 AND "Unit1.Em4.ControlNodes".ngPnP."step".transition1[240],
                         PT := #delayTime);
   IF #statTonTime[240].Q THEN
       "Unit1.Em4.ControlNodes".ngPnP.sequence.status.nextStep := #JOB_2_STEP_80;
   END_IF;
END_REGION

REGION Network 21: Step[280] : NG P&P 1,2 Backward
   RUNG wire#powerrail
      { S7_Templates := "SrcType := DInt" } EQ_Contact(in1 := "Unit1.Em4.ControlNodes".ngPnP.sequence.status.currentStep, in2 := #JOB_2_STEP_80)
      Contact( "Unit1.Em4.ControlNodes".ngPnP.sequence.status.seqActive )
      wire#w1
      I_Contact( "Unit1.Em4.ControlNodes".cmAnodeNgPnp1stFwdBwd.monitoring.inHomePos )
      wire#w2
      Coil( "Unit1.Em4.ControlNodes".ngPnP."step".action1[280] )
   END_RUNG
   RUNG wire#w1
      I_Contact( "Unit1.Em4.ControlNodes".cmAnodeNgPnp2ndFwdBwd.monitoring.inHomePos )
   END_RUNG wire#w2
   RUNG wire#w1
      Contact( "Unit1.Em4.ControlNodes".cmAnodeNgPnp1stFwdBwd.monitoring.inHomePos )
      Contact( "Unit1.Em4.ControlNodes".cmAnodeNgPnp2ndFwdBwd.monitoring.inHomePos )
      Contact( "Unit1.Em4.ControlNodes".cm.softCam.anodeAlignTableAxisX.waitPos.inPos )
      Contact( "Unit1.Em4.ControlNodes".cm.softCam.anodeAlignTableAxisY1.waitPos.inPos )
      Contact( "Unit1.Em4.ControlNodes".cm.softCam.anodeAlignTableAxisY2.waitPos.inPos )
      Coil( "Unit1.Em4.ControlNodes".ngPnP."step".transition1[280] )
   END_RUNG
   RUNG wire#w1
      Contact( "Unit1.Em4.ControlNodes".ngPnP."step".transition1[280] )
      { S7_Templates := "time_type := Time" } #statTonTime[280].TON(pt := #delayTime, et =>)
      Move(in := #JOB_2_STEP_90, out1 => "Unit1.Em4.ControlNodes".ngPnP.sequence.status.nextStep)
   END_RUNG
   // the same network as SCL:
   #_w1 := ("Unit1.Em4.ControlNodes".ngPnP.sequence.status.currentStep = #JOB_2_STEP_80) AND "Unit1.Em4.ControlNodes".ngPnP.sequence.status.seqActive;
   "Unit1.Em4.ControlNodes".ngPnP."step".action1[280] := #_w1 AND (NOT "Unit1.Em4.ControlNodes".cmAnodeNgPnp1stFwdBwd.monitoring.inHomePos OR NOT "Unit1.Em4.ControlNodes".cmAnodeNgPnp2ndFwdBwd.monitoring.inHomePos);
   "Unit1.Em4.ControlNodes".ngPnP."step".transition1[280] := #_w1 AND "Unit1.Em4.ControlNodes".cmAnodeNgPnp1stFwdBwd.monitoring.inHomePos AND "Unit1.Em4.ControlNodes".cmAnodeNgPnp2ndFwdBwd.monitoring.inHomePos AND "Unit1.Em4.ControlNodes".cm.softCam.anodeAlignTableAxisX.waitPos.inPos AND "Unit1.Em4.ControlNodes".cm.softCam.anodeAlignTableAxisY1.waitPos.inPos AND "Unit1.Em4.ControlNodes".cm.softCam.anodeAlignTableAxisY2.waitPos.inPos;
   #statTonTime[280].TON(IN := #_w1 AND "Unit1.Em4.ControlNodes".ngPnP."step".transition1[280],
                         PT := #delayTime);
   IF #statTonTime[280].Q THEN
       "Unit1.Em4.ControlNodes".ngPnP.sequence.status.nextStep := #JOB_2_STEP_90;
   END_IF;
END_REGION

REGION Network 22: Step[290] : JOB[2] Condition
   RUNG wire#powerrail
      { S7_Templates := "SrcType := DInt" } EQ_Contact(in1 := "Unit1.Em4.ControlNodes".ngPnP.sequence.status.currentStep, in2 := #JOB_2_STEP_90)
      Contact( "Unit1.Em4.ControlNodes".ngPnP.sequence.status.seqActive )
      wire#w1
      Coil( "Unit1.Em4.ControlNodes".ngPnP."step".action1[290] )
   END_RUNG
   RUNG wire#w1
      Coil( "Unit1.Em4.ControlNodes".ngPnP."step".transition1[290] )
   END_RUNG
   RUNG wire#w1
      Contact( "Unit1.Em4.ControlNodes".ngPnP."step".transition1[290] )
      { S7_Templates := "time_type := Time" } #statTonTime[290].TON(pt := #delayTime, et =>)
      Move(in := #STEP_IDLE, out1 => "Unit1.Em4.ControlNodes".ngPnP.sequence.status.nextStep)
   END_RUNG
   // the same network as SCL:
   "Unit1.Em4.ControlNodes".ngPnP."step".action1[290] := ("Unit1.Em4.ControlNodes".ngPnP.sequence.status.currentStep = #JOB_2_STEP_90) AND "Unit1.Em4.ControlNodes".ngPnP.sequence.status.seqActive;
   "Unit1.Em4.ControlNodes".ngPnP."step".transition1[290] := ("Unit1.Em4.ControlNodes".ngPnP.sequence.status.currentStep = #JOB_2_STEP_90) AND "Unit1.Em4.ControlNodes".ngPnP.sequence.status.seqActive;
   #statTonTime[290].TON(IN := ("Unit1.Em4.ControlNodes".ngPnP.sequence.status.currentStep = #JOB_2_STEP_90) AND "Unit1.Em4.ControlNodes".ngPnP.sequence.status.seqActive AND "Unit1.Em4.ControlNodes".ngPnP."step".transition1[290],
                         PT := #delayTime);
   IF #statTonTime[290].Q THEN "Unit1.Em4.ControlNodes".ngPnP.sequence.status.nextStep := #STEP_IDLE; END_IF;
END_REGION

REGION Network 23: *************** JOB[3] Unloading ************************
END_REGION

REGION Network 24: Step[301] : JOB[3] Condition
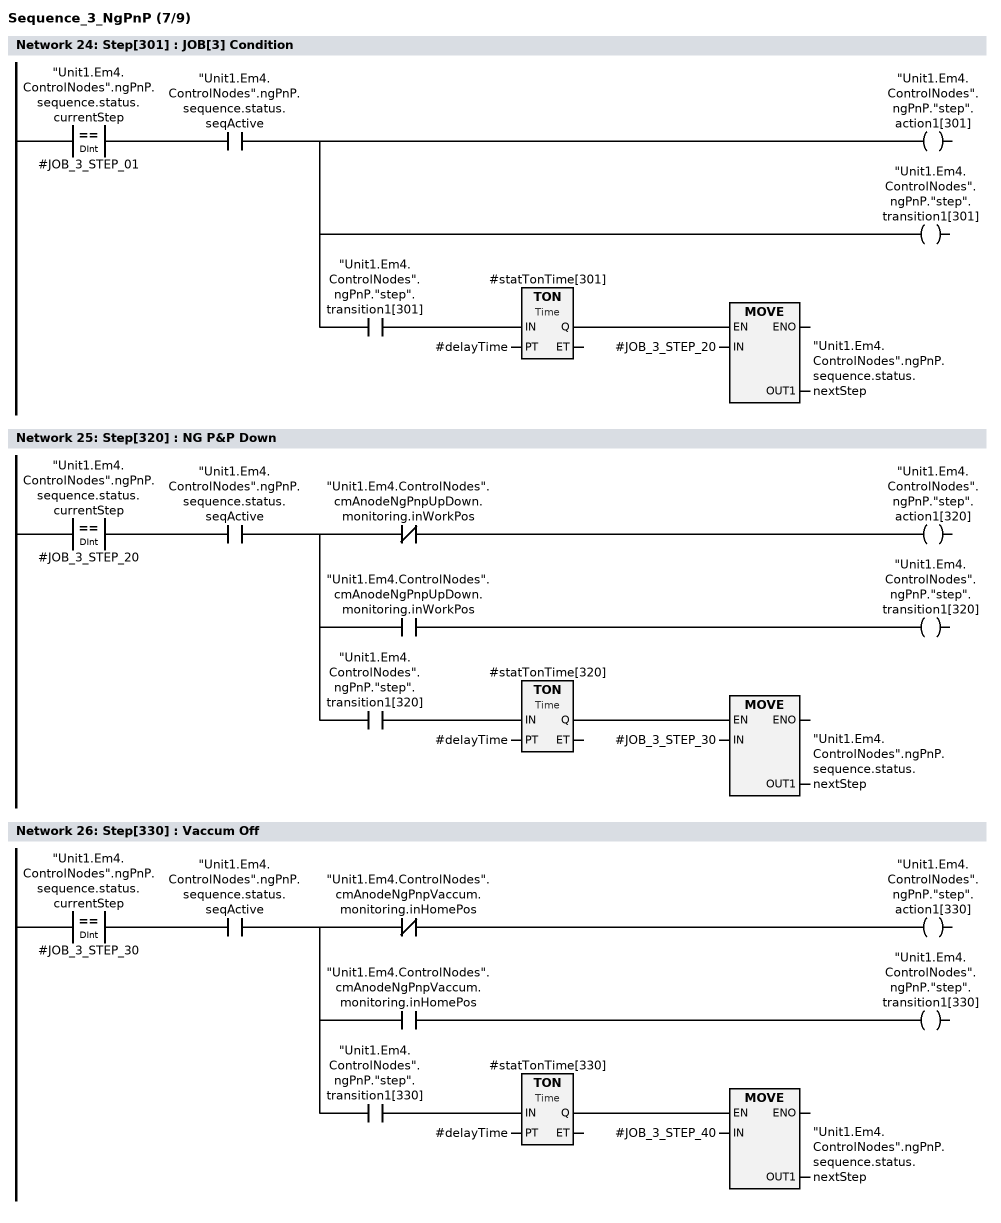
   RUNG wire#powerrail
      { S7_Templates := "SrcType := DInt" } EQ_Contact(in1 := "Unit1.Em4.ControlNodes".ngPnP.sequence.status.currentStep, in2 := #JOB_3_STEP_01)
      Contact( "Unit1.Em4.ControlNodes".ngPnP.sequence.status.seqActive )
      wire#w1
      Coil( "Unit1.Em4.ControlNodes".ngPnP."step".action1[301] )
   END_RUNG
   RUNG wire#w1
      Coil( "Unit1.Em4.ControlNodes".ngPnP."step".transition1[301] )
   END_RUNG
   RUNG wire#w1
      Contact( "Unit1.Em4.ControlNodes".ngPnP."step".transition1[301] )
      { S7_Templates := "time_type := Time" } #statTonTime[301].TON(pt := #delayTime, et =>)
      Move(in := #JOB_3_STEP_20, out1 => "Unit1.Em4.ControlNodes".ngPnP.sequence.status.nextStep)
   END_RUNG
   // the same network as SCL:
   "Unit1.Em4.ControlNodes".ngPnP."step".action1[301] := ("Unit1.Em4.ControlNodes".ngPnP.sequence.status.currentStep = #JOB_3_STEP_01) AND "Unit1.Em4.ControlNodes".ngPnP.sequence.status.seqActive;
   "Unit1.Em4.ControlNodes".ngPnP."step".transition1[301] := ("Unit1.Em4.ControlNodes".ngPnP.sequence.status.currentStep = #JOB_3_STEP_01) AND "Unit1.Em4.ControlNodes".ngPnP.sequence.status.seqActive;
   #statTonTime[301].TON(IN := ("Unit1.Em4.ControlNodes".ngPnP.sequence.status.currentStep = #JOB_3_STEP_01) AND "Unit1.Em4.ControlNodes".ngPnP.sequence.status.seqActive AND "Unit1.Em4.ControlNodes".ngPnP."step".transition1[301],
                         PT := #delayTime);
   IF #statTonTime[301].Q THEN
       "Unit1.Em4.ControlNodes".ngPnP.sequence.status.nextStep := #JOB_3_STEP_20;
   END_IF;
END_REGION

REGION Network 25: Step[320] : NG P&P Down
   RUNG wire#powerrail
      { S7_Templates := "SrcType := DInt" } EQ_Contact(in1 := "Unit1.Em4.ControlNodes".ngPnP.sequence.status.currentStep, in2 := #JOB_3_STEP_20)
      Contact( "Unit1.Em4.ControlNodes".ngPnP.sequence.status.seqActive )
      wire#w1
      I_Contact( "Unit1.Em4.ControlNodes".cmAnodeNgPnpUpDown.monitoring.inWorkPos )
      Coil( "Unit1.Em4.ControlNodes".ngPnP."step".action1[320] )
   END_RUNG
   RUNG wire#w1
      Contact( "Unit1.Em4.ControlNodes".cmAnodeNgPnpUpDown.monitoring.inWorkPos )
      Coil( "Unit1.Em4.ControlNodes".ngPnP."step".transition1[320] )
   END_RUNG
   RUNG wire#w1
      Contact( "Unit1.Em4.ControlNodes".ngPnP."step".transition1[320] )
      { S7_Templates := "time_type := Time" } #statTonTime[320].TON(pt := #delayTime, et =>)
      Move(in := #JOB_3_STEP_30, out1 => "Unit1.Em4.ControlNodes".ngPnP.sequence.status.nextStep)
   END_RUNG
   // the same network as SCL:
   #_w1 := ("Unit1.Em4.ControlNodes".ngPnP.sequence.status.currentStep = #JOB_3_STEP_20) AND "Unit1.Em4.ControlNodes".ngPnP.sequence.status.seqActive;
   "Unit1.Em4.ControlNodes".ngPnP."step".action1[320] := #_w1 AND NOT "Unit1.Em4.ControlNodes".cmAnodeNgPnpUpDown.monitoring.inWorkPos;
   "Unit1.Em4.ControlNodes".ngPnP."step".transition1[320] := #_w1 AND "Unit1.Em4.ControlNodes".cmAnodeNgPnpUpDown.monitoring.inWorkPos;
   #statTonTime[320].TON(IN := #_w1 AND "Unit1.Em4.ControlNodes".ngPnP."step".transition1[320],
                         PT := #delayTime);
   IF #statTonTime[320].Q THEN
       "Unit1.Em4.ControlNodes".ngPnP.sequence.status.nextStep := #JOB_3_STEP_30;
   END_IF;
END_REGION

REGION Network 26: Step[330] : Vaccum Off
   RUNG wire#powerrail
      { S7_Templates := "SrcType := DInt" } EQ_Contact(in1 := "Unit1.Em4.ControlNodes".ngPnP.sequence.status.currentStep, in2 := #JOB_3_STEP_30)
      Contact( "Unit1.Em4.ControlNodes".ngPnP.sequence.status.seqActive )
      wire#w1
      I_Contact( "Unit1.Em4.ControlNodes".cmAnodeNgPnpVaccum.monitoring.inHomePos )
      Coil( "Unit1.Em4.ControlNodes".ngPnP."step".action1[330] )
   END_RUNG
   RUNG wire#w1
      Contact( "Unit1.Em4.ControlNodes".cmAnodeNgPnpVaccum.monitoring.inHomePos )
      Coil( "Unit1.Em4.ControlNodes".ngPnP."step".transition1[330] )
   END_RUNG
   RUNG wire#w1
      Contact( "Unit1.Em4.ControlNodes".ngPnP."step".transition1[330] )
      { S7_Templates := "time_type := Time" } #statTonTime[330].TON(pt := #delayTime, et =>)
      Move(in := #JOB_3_STEP_40, out1 => "Unit1.Em4.ControlNodes".ngPnP.sequence.status.nextStep)
   END_RUNG
   // the same network as SCL:
   #_w1 := ("Unit1.Em4.ControlNodes".ngPnP.sequence.status.currentStep = #JOB_3_STEP_30) AND "Unit1.Em4.ControlNodes".ngPnP.sequence.status.seqActive;
   "Unit1.Em4.ControlNodes".ngPnP."step".action1[330] := #_w1 AND NOT "Unit1.Em4.ControlNodes".cmAnodeNgPnpVaccum.monitoring.inHomePos;
   "Unit1.Em4.ControlNodes".ngPnP."step".transition1[330] := #_w1 AND "Unit1.Em4.ControlNodes".cmAnodeNgPnpVaccum.monitoring.inHomePos;
   #statTonTime[330].TON(IN := #_w1 AND "Unit1.Em4.ControlNodes".ngPnP."step".transition1[330],
                         PT := #delayTime);
   IF #statTonTime[330].Q THEN
       "Unit1.Em4.ControlNodes".ngPnP.sequence.status.nextStep := #JOB_3_STEP_40;
   END_IF;
END_REGION

REGION Network 27: Step[340] : NG P&P Up
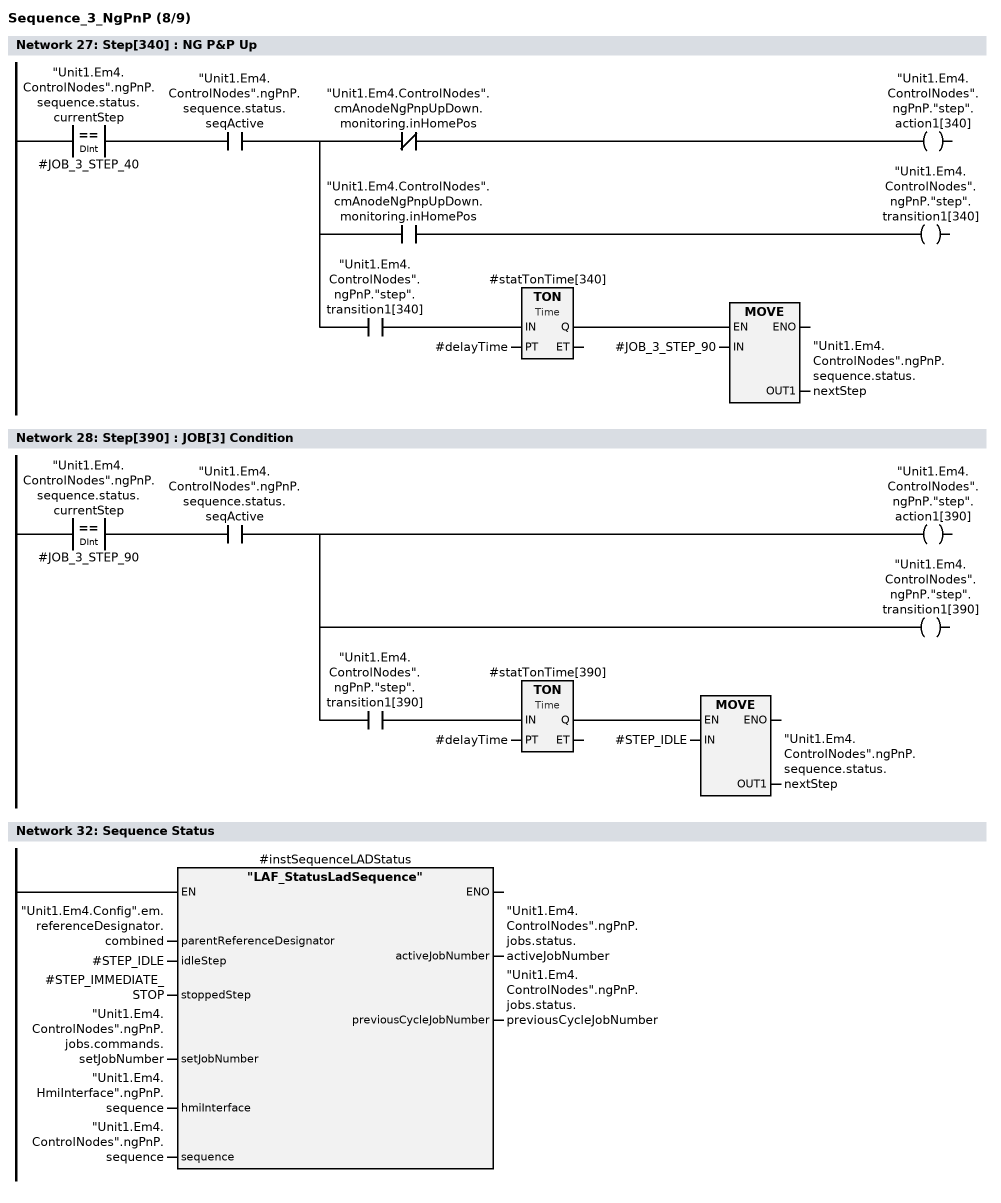
   RUNG wire#powerrail
      { S7_Templates := "SrcType := DInt" } EQ_Contact(in1 := "Unit1.Em4.ControlNodes".ngPnP.sequence.status.currentStep, in2 := #JOB_3_STEP_40)
      Contact( "Unit1.Em4.ControlNodes".ngPnP.sequence.status.seqActive )
      wire#w1
      I_Contact( "Unit1.Em4.ControlNodes".cmAnodeNgPnpUpDown.monitoring.inHomePos )
      Coil( "Unit1.Em4.ControlNodes".ngPnP."step".action1[340] )
   END_RUNG
   RUNG wire#w1
      Contact( "Unit1.Em4.ControlNodes".cmAnodeNgPnpUpDown.monitoring.inHomePos )
      Coil( "Unit1.Em4.ControlNodes".ngPnP."step".transition1[340] )
   END_RUNG
   RUNG wire#w1
      Contact( "Unit1.Em4.ControlNodes".ngPnP."step".transition1[340] )
      { S7_Templates := "time_type := Time" } #statTonTime[340].TON(pt := #delayTime, et =>)
      Move(in := #JOB_3_STEP_90, out1 => "Unit1.Em4.ControlNodes".ngPnP.sequence.status.nextStep)
   END_RUNG
   // the same network as SCL:
   #_w1 := ("Unit1.Em4.ControlNodes".ngPnP.sequence.status.currentStep = #JOB_3_STEP_40) AND "Unit1.Em4.ControlNodes".ngPnP.sequence.status.seqActive;
   "Unit1.Em4.ControlNodes".ngPnP."step".action1[340] := #_w1 AND NOT "Unit1.Em4.ControlNodes".cmAnodeNgPnpUpDown.monitoring.inHomePos;
   "Unit1.Em4.ControlNodes".ngPnP."step".transition1[340] := #_w1 AND "Unit1.Em4.ControlNodes".cmAnodeNgPnpUpDown.monitoring.inHomePos;
   #statTonTime[340].TON(IN := #_w1 AND "Unit1.Em4.ControlNodes".ngPnP."step".transition1[340],
                         PT := #delayTime);
   IF #statTonTime[340].Q THEN
       "Unit1.Em4.ControlNodes".ngPnP.sequence.status.nextStep := #JOB_3_STEP_90;
   END_IF;
END_REGION

REGION Network 28: Step[390] : JOB[3] Condition
   RUNG wire#powerrail
      { S7_Templates := "SrcType := DInt" } EQ_Contact(in1 := "Unit1.Em4.ControlNodes".ngPnP.sequence.status.currentStep, in2 := #JOB_3_STEP_90)
      Contact( "Unit1.Em4.ControlNodes".ngPnP.sequence.status.seqActive )
      wire#w1
      Coil( "Unit1.Em4.ControlNodes".ngPnP."step".action1[390] )
   END_RUNG
   RUNG wire#w1
      Coil( "Unit1.Em4.ControlNodes".ngPnP."step".transition1[390] )
   END_RUNG
   RUNG wire#w1
      Contact( "Unit1.Em4.ControlNodes".ngPnP."step".transition1[390] )
      { S7_Templates := "time_type := Time" } #statTonTime[390].TON(pt := #delayTime, et =>)
      Move(in := #STEP_IDLE, out1 => "Unit1.Em4.ControlNodes".ngPnP.sequence.status.nextStep)
   END_RUNG
   // the same network as SCL:
   "Unit1.Em4.ControlNodes".ngPnP."step".action1[390] := ("Unit1.Em4.ControlNodes".ngPnP.sequence.status.currentStep = #JOB_3_STEP_90) AND "Unit1.Em4.ControlNodes".ngPnP.sequence.status.seqActive;
   "Unit1.Em4.ControlNodes".ngPnP."step".transition1[390] := ("Unit1.Em4.ControlNodes".ngPnP.sequence.status.currentStep = #JOB_3_STEP_90) AND "Unit1.Em4.ControlNodes".ngPnP.sequence.status.seqActive;
   #statTonTime[390].TON(IN := ("Unit1.Em4.ControlNodes".ngPnP.sequence.status.currentStep = #JOB_3_STEP_90) AND "Unit1.Em4.ControlNodes".ngPnP.sequence.status.seqActive AND "Unit1.Em4.ControlNodes".ngPnP."step".transition1[390],
                         PT := #delayTime);
   IF #statTonTime[390].Q THEN "Unit1.Em4.ControlNodes".ngPnP.sequence.status.nextStep := #STEP_IDLE; END_IF;
END_REGION

REGION Network 29: *************** IMMEDIATE STOP **************************
END_REGION

REGION Network 30: Immediate Stop
END_REGION

REGION Network 31: *************** Status updates **************************
END_REGION

REGION Network 32: Sequence Status
   RUNG wire#powerrail
      #instSequenceLADStatus(parentReferenceDesignator := "Unit1.Em4.Config".em.referenceDesignator.combined, idleStep := #STEP_IDLE, stoppedStep := #STEP_IMMEDIATE_STOP, setJobNumber := "Unit1.Em4.ControlNodes".ngPnP.jobs.commands.setJobNumber, hmiInterface := "Unit1.Em4.HmiInterface".ngPnP.sequence, sequence := "Unit1.Em4.ControlNodes".ngPnP.sequence, activeJobNumber => "Unit1.Em4.ControlNodes".ngPnP.jobs.status.activeJobNumber, previousCycleJobNumber => "Unit1.Em4.ControlNodes".ngPnP.jobs.status.previousCycleJobNumber)
   END_RUNG
   // the same network as SCL:
   #instSequenceLADStatus(parentReferenceDesignator := "Unit1.Em4.Config".em.referenceDesignator.combined,   // "LAF_StatusLadSequence"
                          idleStep := #STEP_IDLE,
                          stoppedStep := #STEP_IMMEDIATE_STOP,
                          setJobNumber := "Unit1.Em4.ControlNodes".ngPnP.jobs.commands.setJobNumber,
                          hmiInterface := "Unit1.Em4.HmiInterface".ngPnP.sequence,
                          sequence := "Unit1.Em4.ControlNodes".ngPnP.sequence,
                          activeJobNumber => "Unit1.Em4.ControlNodes".ngPnP.jobs.status.activeJobNumber,
                          previousCycleJobNumber => "Unit1.Em4.ControlNodes".ngPnP.jobs.status.previousCycleJobNumber);
END_REGION

REGION Network 33: Update Job History
   // Update the History of jobs if a new job was started
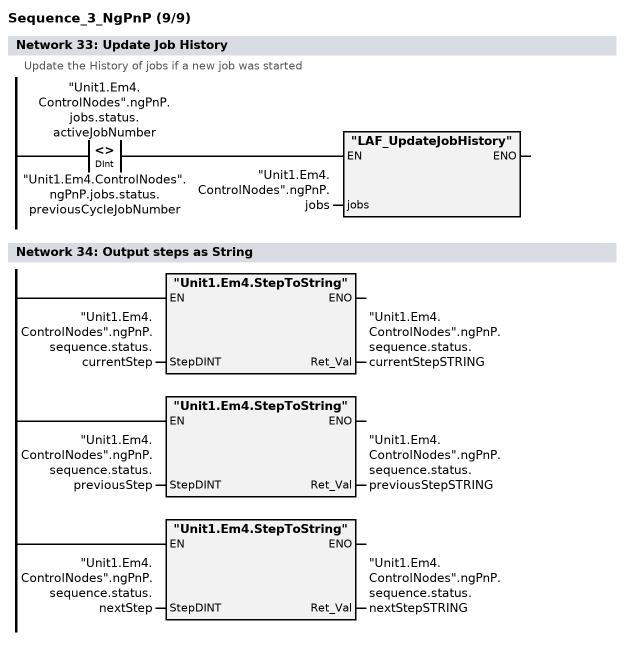
   RUNG wire#powerrail
      { S7_Templates := "SrcType := DInt" } NE_Contact(in1 := "Unit1.Em4.ControlNodes".ngPnP.jobs.status.activeJobNumber, in2 := "Unit1.Em4.ControlNodes".ngPnP.jobs.status.previousCycleJobNumber)
      "LAF_UpdateJobHistory"(jobs := "Unit1.Em4.ControlNodes".ngPnP.jobs)
   END_RUNG
   // the same network as SCL:
   IF "Unit1.Em4.ControlNodes".ngPnP.jobs.status.activeJobNumber <> "Unit1.Em4.ControlNodes".ngPnP.jobs.status.previousCycleJobNumber THEN
       "LAF_UpdateJobHistory"(jobs := "Unit1.Em4.ControlNodes".ngPnP.jobs);
   END_IF;
END_REGION

REGION Network 34: Output steps as String
   RUNG wire#powerrail
      "Unit1.Em4.StepToString"(StepDINT := "Unit1.Em4.ControlNodes".ngPnP.sequence.status.currentStep, Ret_Val => "Unit1.Em4.ControlNodes".ngPnP.sequence.status.currentStepSTRING)
   END_RUNG
   RUNG wire#powerrail
      "Unit1.Em4.StepToString"(StepDINT := "Unit1.Em4.ControlNodes".ngPnP.sequence.status.previousStep, Ret_Val => "Unit1.Em4.ControlNodes".ngPnP.sequence.status.previousStepSTRING)
   END_RUNG
   RUNG wire#powerrail
      "Unit1.Em4.StepToString"(StepDINT := "Unit1.Em4.ControlNodes".ngPnP.sequence.status.nextStep, Ret_Val => "Unit1.Em4.ControlNodes".ngPnP.sequence.status.nextStepSTRING)
   END_RUNG
   // the same network as SCL:
   "Unit1.Em4.ControlNodes".ngPnP.sequence.status.currentStepSTRING := "Unit1.Em4.StepToString"(StepDINT := "Unit1.Em4.ControlNodes".ngPnP.sequence.status.currentStep);
   "Unit1.Em4.ControlNodes".ngPnP.sequence.status.previousStepSTRING := "Unit1.Em4.StepToString"(StepDINT := "Unit1.Em4.ControlNodes".ngPnP.sequence.status.previousStep);
   "Unit1.Em4.ControlNodes".ngPnP.sequence.status.nextStepSTRING := "Unit1.Em4.StepToString"(StepDINT := "Unit1.Em4.ControlNodes".ngPnP.sequence.status.nextStep);
END_REGION
END_FUNCTION_BLOCK
